(* Logix 5000 project; controller SX_V040001_C001 vendor 1 type 14 code 77 rev 16.22; software revision 16.04; part 18 of 35 *)
(* tags used below, declared in another part *)
   ALL_KINDS : INT[90];
   Basic : INT;
   DRIVE : INT[32];
   Drive_diff_rpm_real : REAL;
   Drive_set_prop_rpm_real : REAL;
   G_AOutput : DINT[8];
   G_DInput : DINT[3];
   G_DOutput : DINT[3];
   PARAMETER : INT[501];
   T_DELAY_COOLING_FAN : TIMER;
   T_DRIVE_START_WARN : TIMER;
   TEMP : INT[14];
(* MainProgram, continued *)

ROUTINE MainDriveFrequenc   (* ladder *)
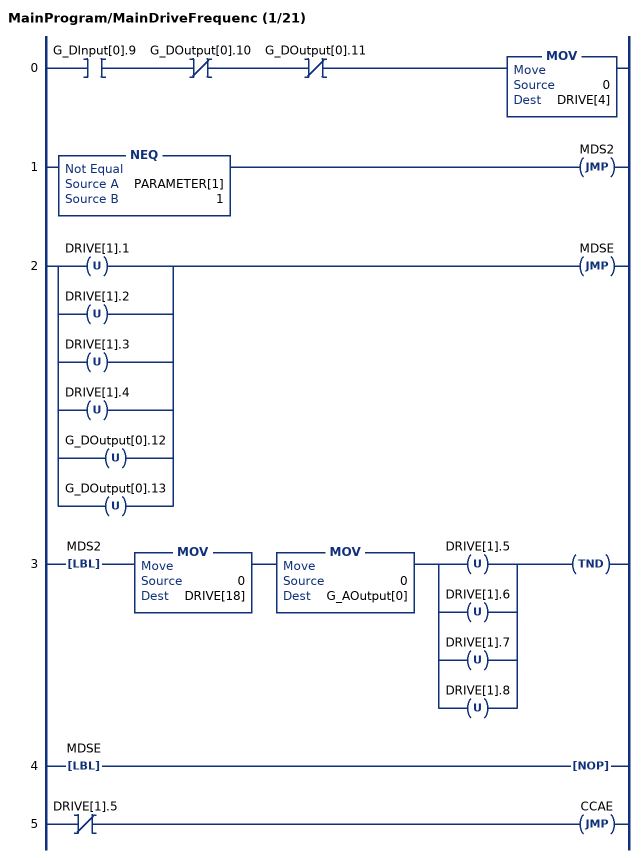
   0: XIC(G_DInput[0].9)XIO(G_DOutput[0].10)XIO(G_DOutput[0].11)MOV(0,DRIVE[4]);
   1: NEQ(PARAMETER[1],1)JMP(MDS2);
   2: [OTU(DRIVE[1].1) ,OTU(DRIVE[1].2) ,OTU(DRIVE[1].3) ,OTU(DRIVE[1].4) ,OTU(G_DOutput[0].12) ,OTU(G_DOutput[0].13) ]JMP(MDSE);
   3: LBL(MDS2)MOV(0,DRIVE[18])MOV(0,G_AOutput[0])[OTU(DRIVE[1].5) ,OTU(DRIVE[1].6) ,OTU(DRIVE[1].7) ,OTU(DRIVE[1].8) ]TND();
   4: LBL(MDSE)NOP();
   5: XIO(DRIVE[1].5)JMP(CCAE);
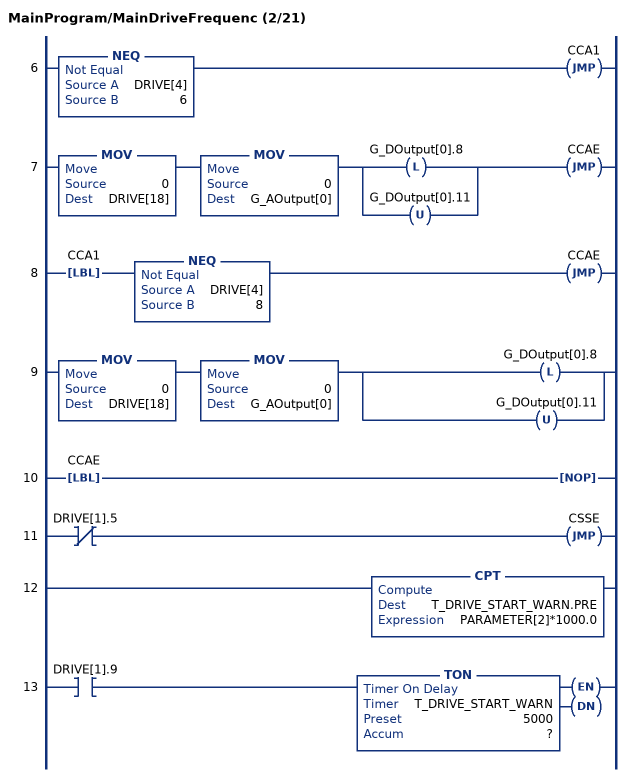
   6: NEQ(DRIVE[4],6)JMP(CCA1);
   7: MOV(0,DRIVE[18])MOV(0,G_AOutput[0])[OTL(G_DOutput[0].8) ,OTU(G_DOutput[0].11) ]JMP(CCAE);
   8: LBL(CCA1)NEQ(DRIVE[4],8)JMP(CCAE);
   9: MOV(0,DRIVE[18])MOV(0,G_AOutput[0])[OTL(G_DOutput[0].8) ,OTU(G_DOutput[0].11) ];
   10: LBL(CCAE)NOP();
   11: XIO(DRIVE[1].5)JMP(CSSE);
   12: CPT(T_DRIVE_START_WARN.PRE,PARAMETER[2]*1000.0);
   13: XIC(DRIVE[1].9)TON(T_DRIVE_START_WARN,?,?);
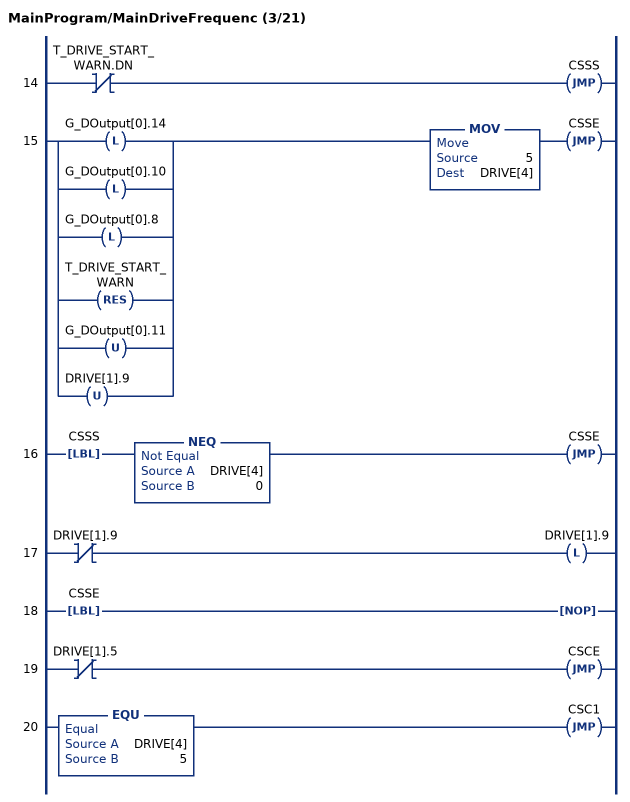
   14: XIO(T_DRIVE_START_WARN.DN)JMP(CSSS);
   15: [OTL(G_DOutput[0].14) ,OTL(G_DOutput[0].10) ,OTL(G_DOutput[0].8) ,RES(T_DRIVE_START_WARN) ,OTU(G_DOutput[0].11) ,OTU(DRIVE[1].9) ]MOV(5,DRIVE[4])JMP(CSSE);
   16: LBL(CSSS)NEQ(DRIVE[4],0)JMP(CSSE);
   17: XIO(DRIVE[1].9)OTL(DRIVE[1].9);
   18: LBL(CSSE)NOP();
   19: XIO(DRIVE[1].5)JMP(CSCE);
   20: EQU(DRIVE[4],5)JMP(CSC1);
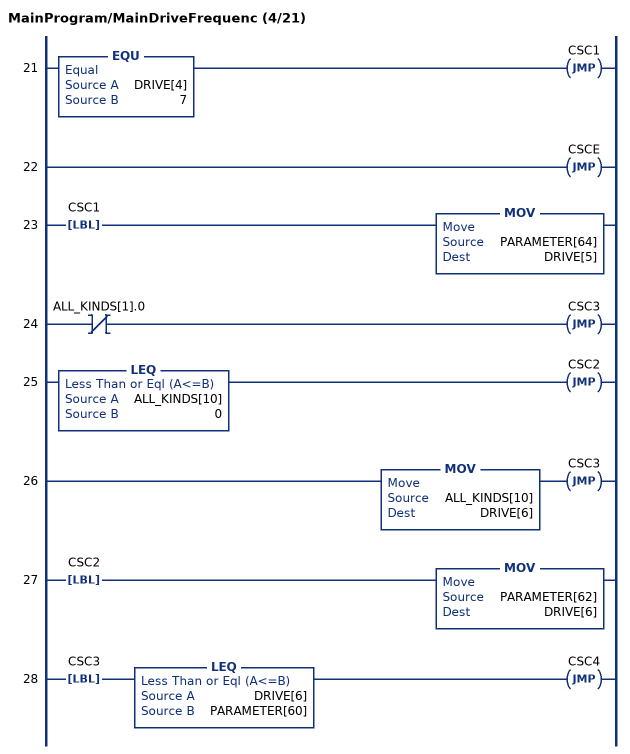
   21: EQU(DRIVE[4],7)JMP(CSC1);
   22: JMP(CSCE);
   23: LBL(CSC1)MOV(PARAMETER[64],DRIVE[5]);
   24: XIO(ALL_KINDS[1].0)JMP(CSC3);
   25: LEQ(ALL_KINDS[10],0)JMP(CSC2);
   26: MOV(ALL_KINDS[10],DRIVE[6])JMP(CSC3);
   27: LBL(CSC2)MOV(PARAMETER[62],DRIVE[6]);
   28: LBL(CSC3)LEQ(DRIVE[6],PARAMETER[60])JMP(CSC4);
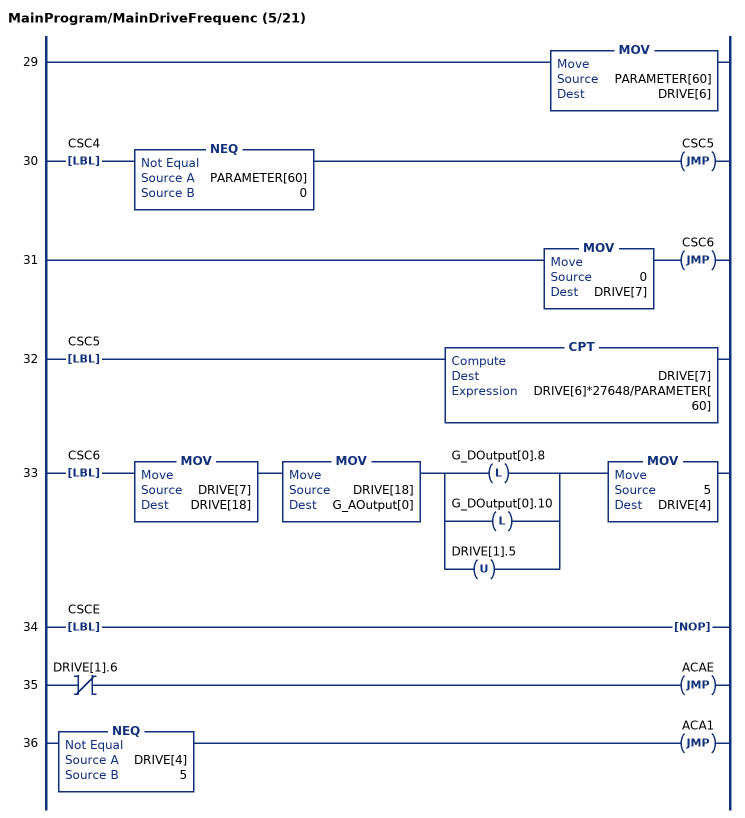
   29: MOV(PARAMETER[60],DRIVE[6]);
   30: LBL(CSC4)NEQ(PARAMETER[60],0)JMP(CSC5);
   31: MOV(0,DRIVE[7])JMP(CSC6);
   32: LBL(CSC5)CPT(DRIVE[7],DRIVE[6]*27648/PARAMETER[60]);
   33: LBL(CSC6)MOV(DRIVE[7],DRIVE[18])MOV(DRIVE[18],G_AOutput[0])[OTL(G_DOutput[0].8) ,OTL(G_DOutput[0].10) ,OTU(DRIVE[1].5) ]MOV(5,DRIVE[4]);
   34: LBL(CSCE)NOP();
   35: XIO(DRIVE[1].6)JMP(ACAE);
   36: NEQ(DRIVE[4],5)JMP(ACA1);
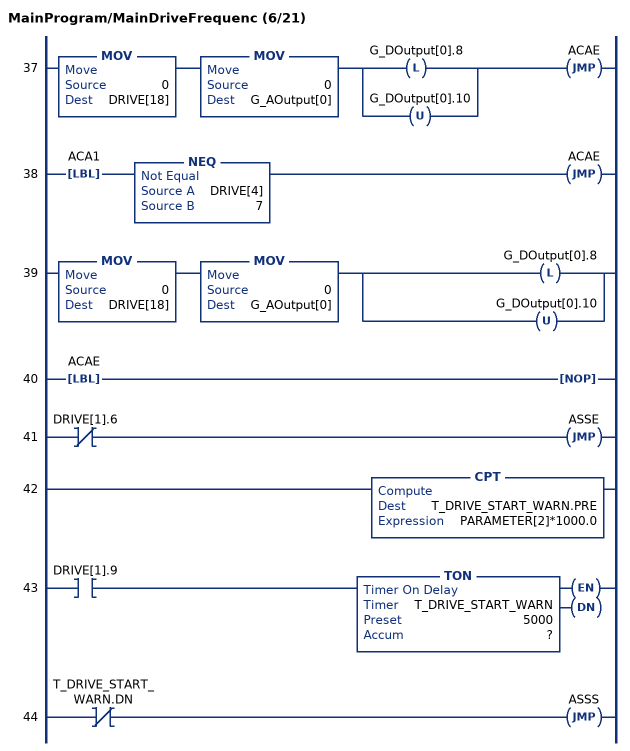
   37: MOV(0,DRIVE[18])MOV(0,G_AOutput[0])[OTL(G_DOutput[0].8) ,OTU(G_DOutput[0].10) ]JMP(ACAE);
   38: LBL(ACA1)NEQ(DRIVE[4],7)JMP(ACAE);
   39: MOV(0,DRIVE[18])MOV(0,G_AOutput[0])[OTL(G_DOutput[0].8) ,OTU(G_DOutput[0].10) ];
   40: LBL(ACAE)NOP();
   41: XIO(DRIVE[1].6)JMP(ASSE);
   42: CPT(T_DRIVE_START_WARN.PRE,PARAMETER[2]*1000.0);
   43: XIC(DRIVE[1].9)TON(T_DRIVE_START_WARN,?,?);
   44: XIO(T_DRIVE_START_WARN.DN)JMP(ASSS);
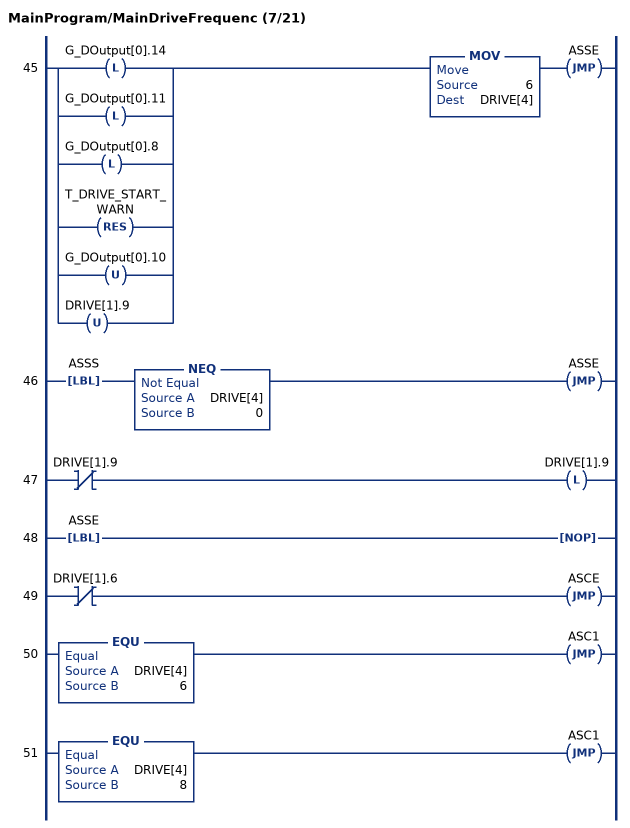
   45: [OTL(G_DOutput[0].14) ,OTL(G_DOutput[0].11) ,OTL(G_DOutput[0].8) ,RES(T_DRIVE_START_WARN) ,OTU(G_DOutput[0].10) ,OTU(DRIVE[1].9) ]MOV(6,DRIVE[4])JMP(ASSE);
   46: LBL(ASSS)NEQ(DRIVE[4],0)JMP(ASSE);
   47: XIO(DRIVE[1].9)OTL(DRIVE[1].9);
   48: LBL(ASSE)NOP();
   49: XIO(DRIVE[1].6)JMP(ASCE);
   50: EQU(DRIVE[4],6)JMP(ASC1);
   51: EQU(DRIVE[4],8)JMP(ASC1);
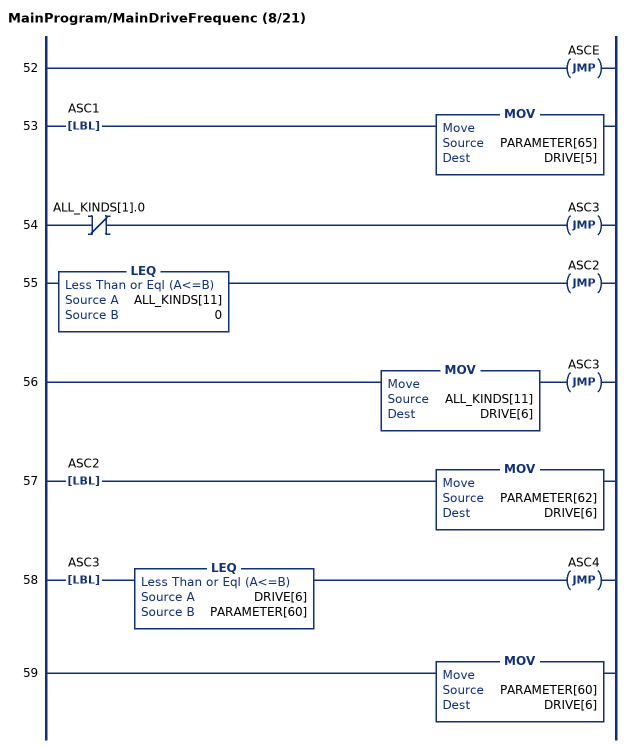
   52: JMP(ASCE);
   53: LBL(ASC1)MOV(PARAMETER[65],DRIVE[5]);
   54: XIO(ALL_KINDS[1].0)JMP(ASC3);
   55: LEQ(ALL_KINDS[11],0)JMP(ASC2);
   56: MOV(ALL_KINDS[11],DRIVE[6])JMP(ASC3);
   57: LBL(ASC2)MOV(PARAMETER[62],DRIVE[6]);
   58: LBL(ASC3)LEQ(DRIVE[6],PARAMETER[60])JMP(ASC4);
   59: MOV(PARAMETER[60],DRIVE[6]);
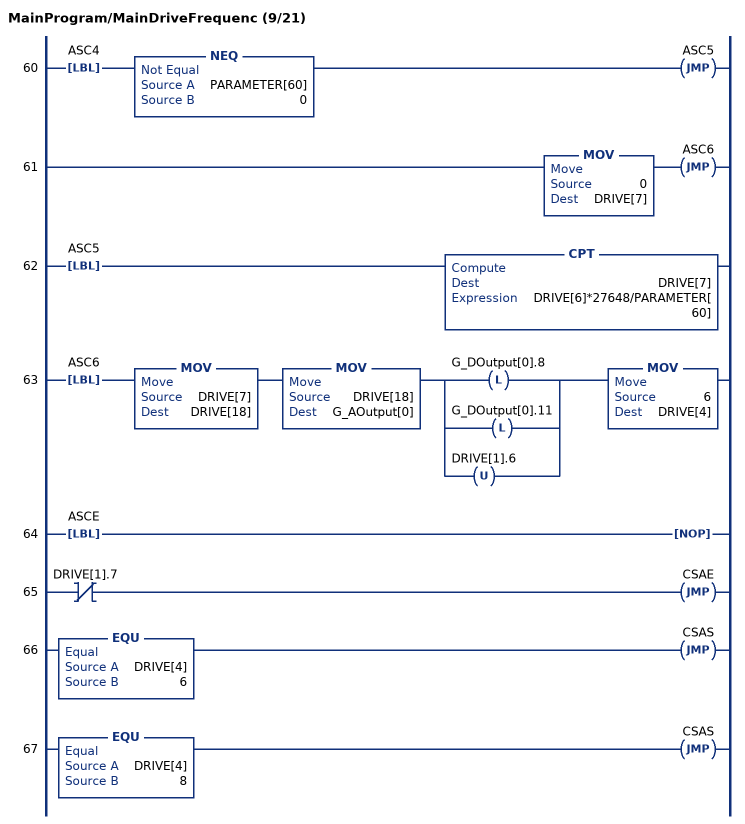
   60: LBL(ASC4)NEQ(PARAMETER[60],0)JMP(ASC5);
   61: MOV(0,DRIVE[7])JMP(ASC6);
   62: LBL(ASC5)CPT(DRIVE[7],DRIVE[6]*27648/PARAMETER[60]);
   63: LBL(ASC6)MOV(DRIVE[7],DRIVE[18])MOV(DRIVE[18],G_AOutput[0])[OTL(G_DOutput[0].8) ,OTL(G_DOutput[0].11) ,OTU(DRIVE[1].6) ]MOV(6,DRIVE[4]);
   64: LBL(ASCE)NOP();
   65: XIO(DRIVE[1].7)JMP(CSAE);
   66: EQU(DRIVE[4],6)JMP(CSAS);
   67: EQU(DRIVE[4],8)JMP(CSAS);
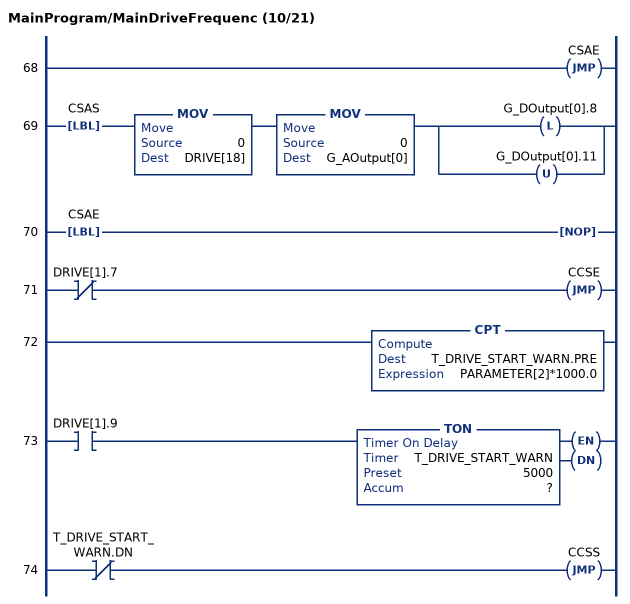
   68: JMP(CSAE);
   69: LBL(CSAS)MOV(0,DRIVE[18])MOV(0,G_AOutput[0])[OTL(G_DOutput[0].8) ,OTU(G_DOutput[0].11) ];
   70: LBL(CSAE)NOP();
   71: XIO(DRIVE[1].7)JMP(CCSE);
   72: CPT(T_DRIVE_START_WARN.PRE,PARAMETER[2]*1000.0);
   73: XIC(DRIVE[1].9)TON(T_DRIVE_START_WARN,?,?);
   74: XIO(T_DRIVE_START_WARN.DN)JMP(CCSS);
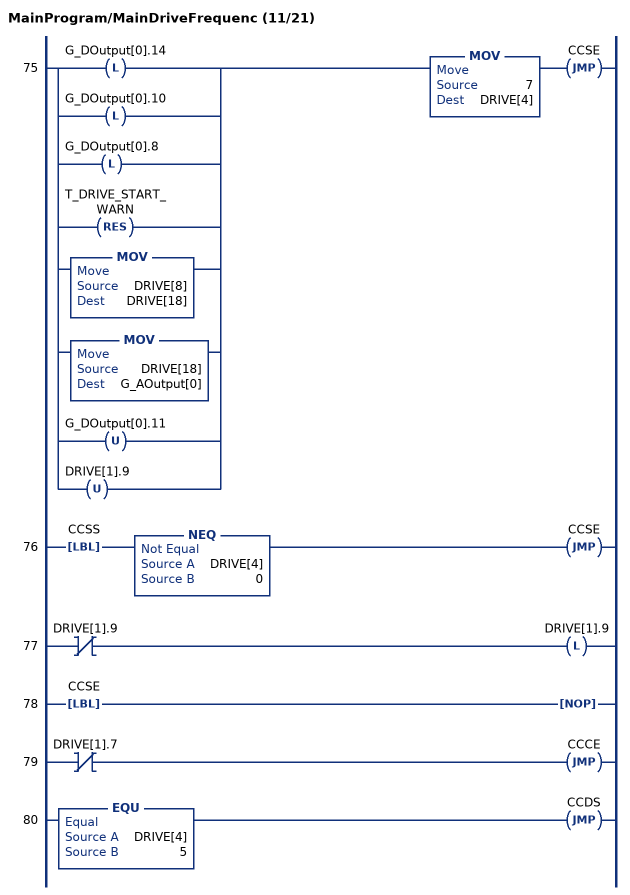
   75: [OTL(G_DOutput[0].14) ,OTL(G_DOutput[0].10) ,OTL(G_DOutput[0].8) ,RES(T_DRIVE_START_WARN) ,MOV(DRIVE[8],DRIVE[18]) ,MOV(DRIVE[18],G_AOutput[0]) ,OTU(G_DOutput[0].11) ,OTU(DRIVE[1].9) ]MOV(7,DRIVE[4])JMP(CCSE);
   76: LBL(CCSS)NEQ(DRIVE[4],0)JMP(CCSE);
   77: XIO(DRIVE[1].9)OTL(DRIVE[1].9);
   78: LBL(CCSE)NOP();
   79: XIO(DRIVE[1].7)JMP(CCCE);
   80: EQU(DRIVE[4],5)JMP(CCDS);
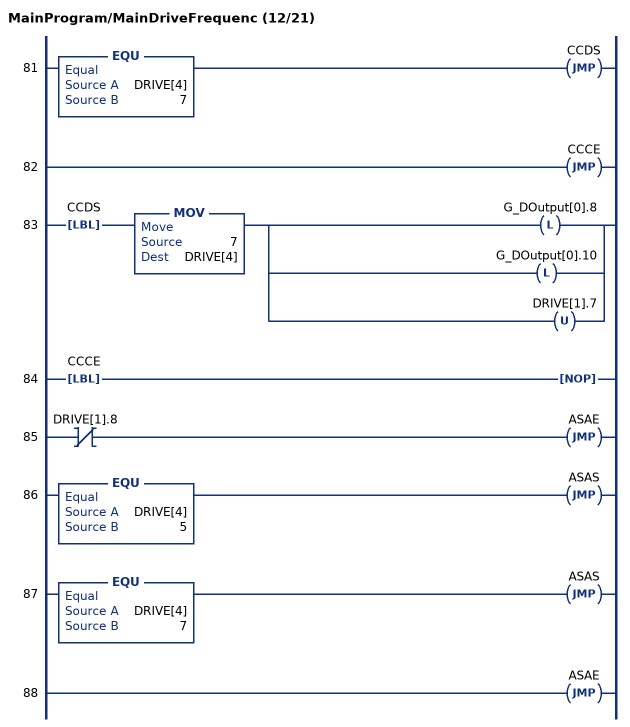
   81: EQU(DRIVE[4],7)JMP(CCDS);
   82: JMP(CCCE);
   83: LBL(CCDS)MOV(7,DRIVE[4])[OTL(G_DOutput[0].8) ,OTL(G_DOutput[0].10) ,OTU(DRIVE[1].7) ];
   84: LBL(CCCE)NOP();
   85: XIO(DRIVE[1].8)JMP(ASAE);
   86: EQU(DRIVE[4],5)JMP(ASAS);
   87: EQU(DRIVE[4],7)JMP(ASAS);
   88: JMP(ASAE);
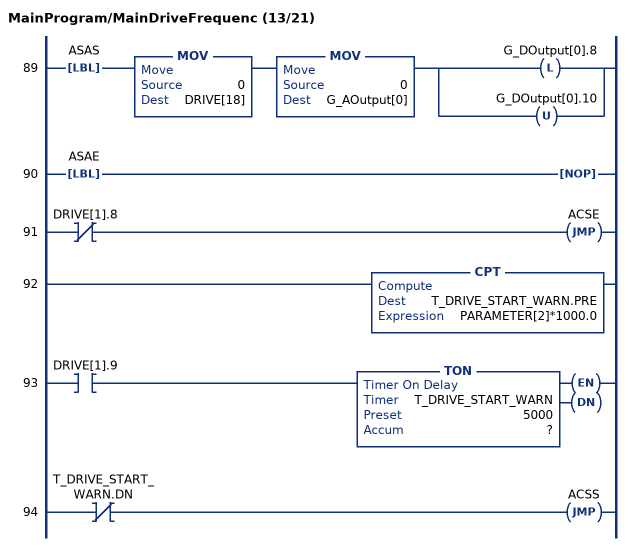
   89: LBL(ASAS)MOV(0,DRIVE[18])MOV(0,G_AOutput[0])[OTL(G_DOutput[0].8) ,OTU(G_DOutput[0].10) ];
   90: LBL(ASAE)NOP();
   91: XIO(DRIVE[1].8)JMP(ACSE);
   92: CPT(T_DRIVE_START_WARN.PRE,PARAMETER[2]*1000.0);
   93: XIC(DRIVE[1].9)TON(T_DRIVE_START_WARN,?,?);
   94: XIO(T_DRIVE_START_WARN.DN)JMP(ACSS);
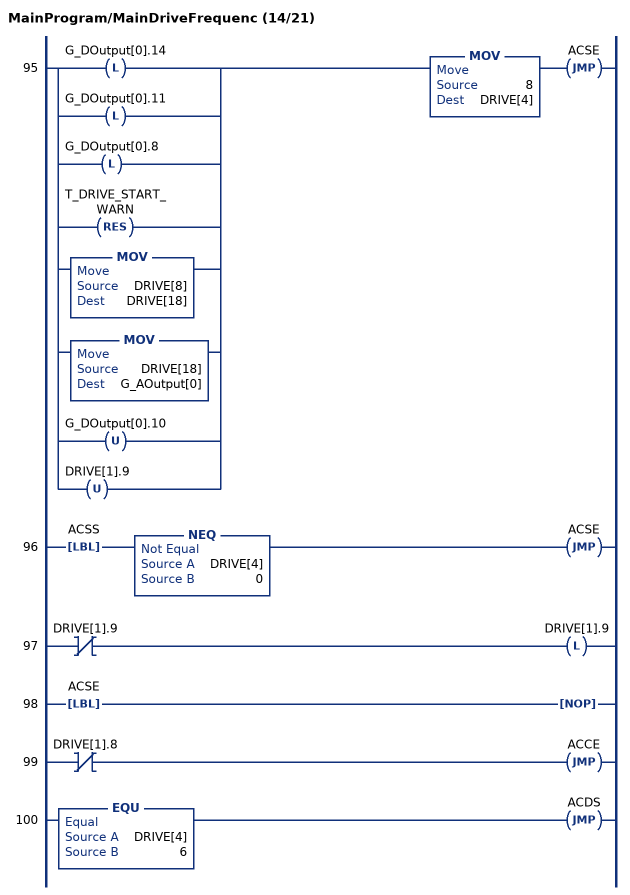
   95: [OTL(G_DOutput[0].14) ,OTL(G_DOutput[0].11) ,OTL(G_DOutput[0].8) ,RES(T_DRIVE_START_WARN) ,MOV(DRIVE[8],DRIVE[18]) ,MOV(DRIVE[18],G_AOutput[0]) ,OTU(G_DOutput[0].10) ,OTU(DRIVE[1].9) ]MOV(8,DRIVE[4])JMP(ACSE);
   96: LBL(ACSS)NEQ(DRIVE[4],0)JMP(ACSE);
   97: XIO(DRIVE[1].9)OTL(DRIVE[1].9);
   98: LBL(ACSE)NOP();
   99: XIO(DRIVE[1].8)JMP(ACCE);
   100: EQU(DRIVE[4],6)JMP(ACDS);
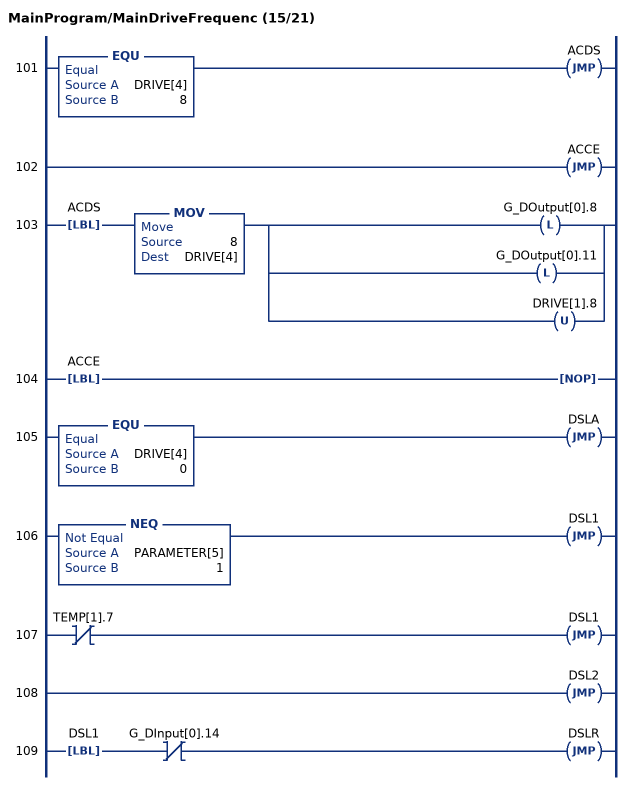
   101: EQU(DRIVE[4],8)JMP(ACDS);
   102: JMP(ACCE);
   103: LBL(ACDS)MOV(8,DRIVE[4])[OTL(G_DOutput[0].8) ,OTL(G_DOutput[0].11) ,OTU(DRIVE[1].8) ];
   104: LBL(ACCE)NOP();
   105: EQU(DRIVE[4],0)JMP(DSLA);
   106: NEQ(PARAMETER[5],1)JMP(DSL1);
   107: XIO(TEMP[1].7)JMP(DSL1);
   108: JMP(DSL2);
   109: LBL(DSL1)XIO(G_DInput[0].14)JMP(DSLR);
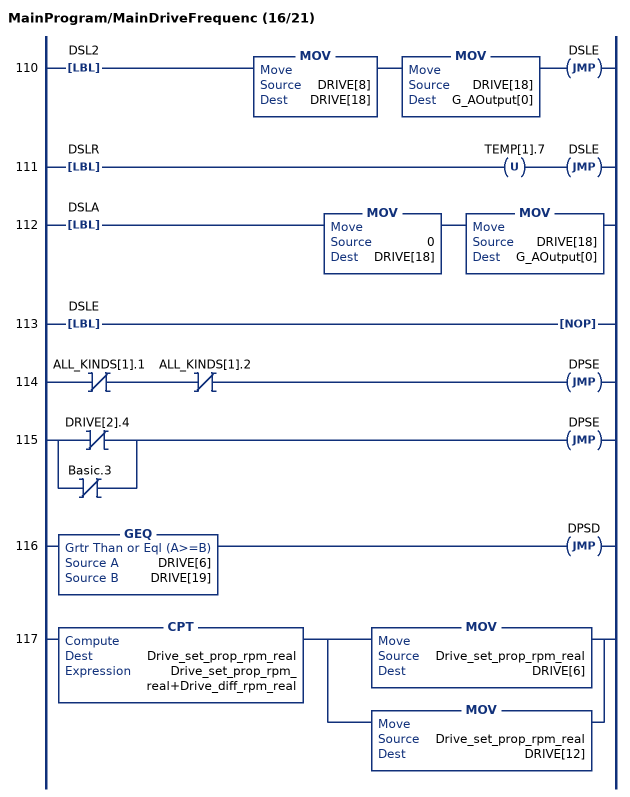
   110: LBL(DSL2)MOV(DRIVE[8],DRIVE[18])MOV(DRIVE[18],G_AOutput[0])JMP(DSLE);
   111: LBL(DSLR)OTU(TEMP[1].7)JMP(DSLE);
   112: LBL(DSLA)MOV(0,DRIVE[18])MOV(DRIVE[18],G_AOutput[0]);
   113: LBL(DSLE)NOP();
   114: XIO(ALL_KINDS[1].1)XIO(ALL_KINDS[1].2)JMP(DPSE);
   115: [XIO(DRIVE[2].4) ,XIO(Basic.3) ]JMP(DPSE);
   116: GEQ(DRIVE[6],DRIVE[19])JMP(DPSD);
   117: CPT(Drive_set_prop_rpm_real,Drive_set_prop_rpm_real+Drive_diff_rpm_real)[MOV(Drive_set_prop_rpm_real,DRIVE[6]) ,MOV(Drive_set_prop_rpm_real,DRIVE[12]) ];
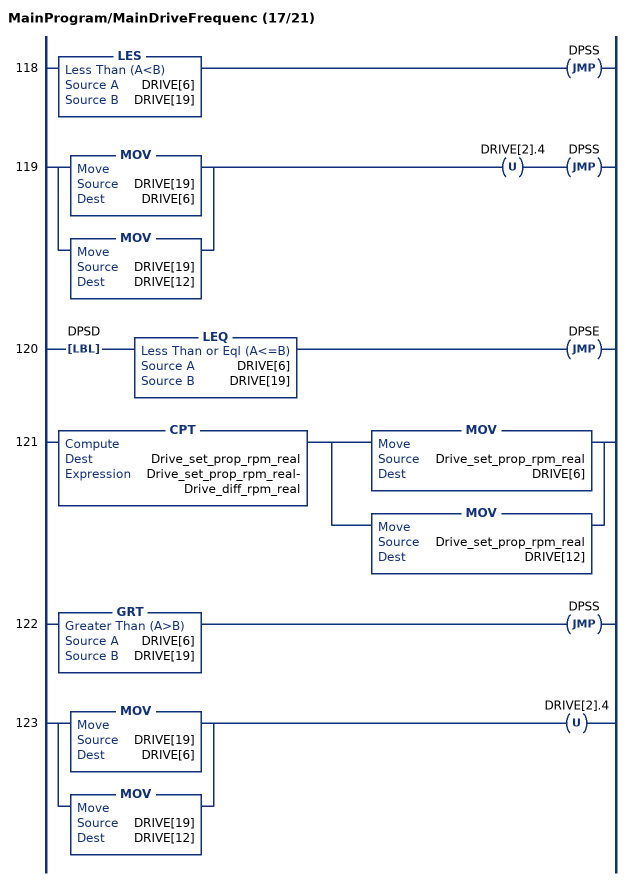
   118: LES(DRIVE[6],DRIVE[19])JMP(DPSS);
   119: [MOV(DRIVE[19],DRIVE[6]) ,MOV(DRIVE[19],DRIVE[12]) ]OTU(DRIVE[2].4)JMP(DPSS);
   120: LBL(DPSD)LEQ(DRIVE[6],DRIVE[19])JMP(DPSE);
   121: CPT(Drive_set_prop_rpm_real,Drive_set_prop_rpm_real-Drive_diff_rpm_real)[MOV(Drive_set_prop_rpm_real,DRIVE[6]) ,MOV(Drive_set_prop_rpm_real,DRIVE[12]) ];
   122: GRT(DRIVE[6],DRIVE[19])JMP(DPSS);
   123: [MOV(DRIVE[19],DRIVE[6]) ,MOV(DRIVE[19],DRIVE[12]) ]OTU(DRIVE[2].4);
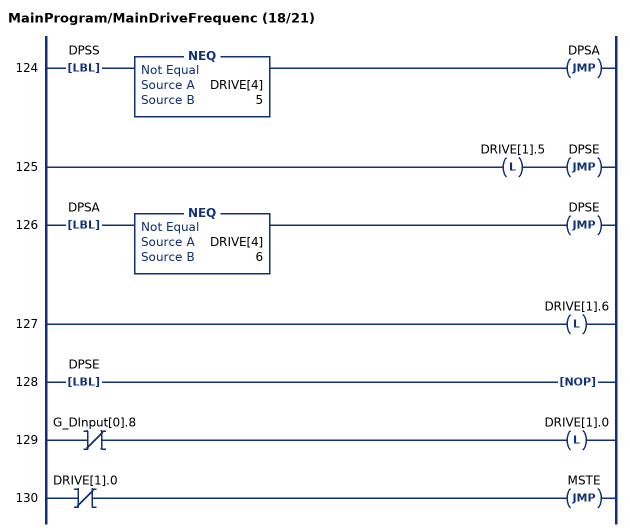
   124: LBL(DPSS)NEQ(DRIVE[4],5)JMP(DPSA);
   125: OTL(DRIVE[1].5)JMP(DPSE);
   126: LBL(DPSA)NEQ(DRIVE[4],6)JMP(DPSE);
   127: OTL(DRIVE[1].6);
   128: LBL(DPSE)NOP();
   129: XIO(G_DInput[0].8)OTL(DRIVE[1].0);
   130: XIO(DRIVE[1].0)JMP(MSTE);
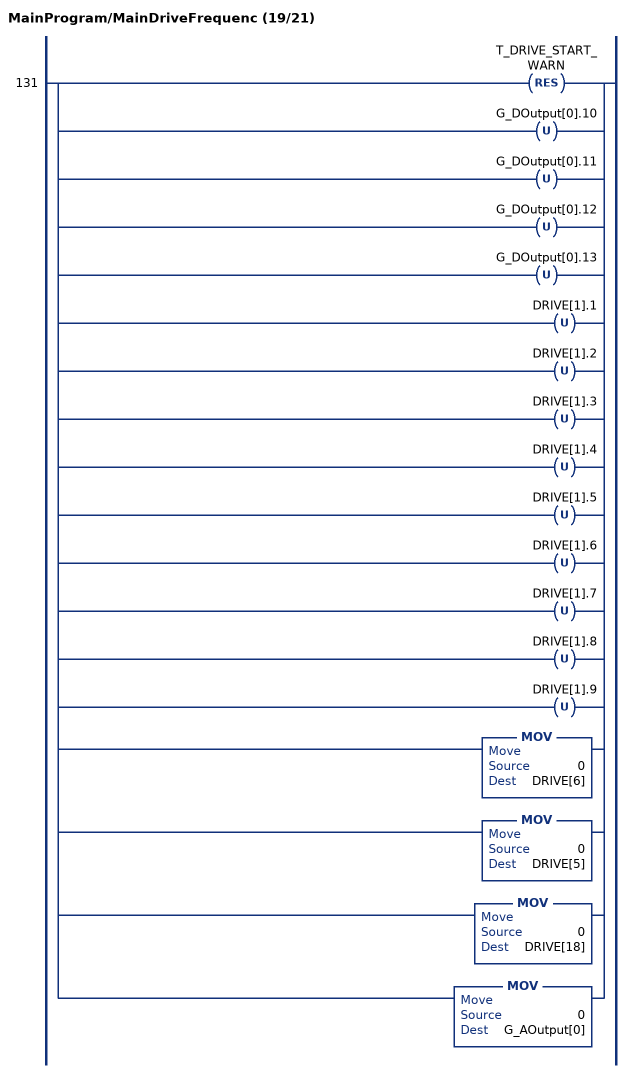
   131: [RES(T_DRIVE_START_WARN) ,OTU(G_DOutput[0].10) ,OTU(G_DOutput[0].11) ,OTU(G_DOutput[0].12) ,OTU(G_DOutput[0].13) ,OTU(DRIVE[1].1) ,OTU(DRIVE[1].2) ,OTU(DRIVE[1].3) ,OTU(DRIVE[1].4) ,OTU(DRIVE[1].5) ,OTU(DRIVE[1].6) ,OTU(DRIVE[1].7) ,OTU(DRIVE[1].8) ,OTU(DRIVE[1].9) ,MOV(0,DRIVE[6]) ,MOV(0,DRIVE[5]) ,MOV(0,DRIVE[18]) ,MOV(0,G_AOutput[0]) ];
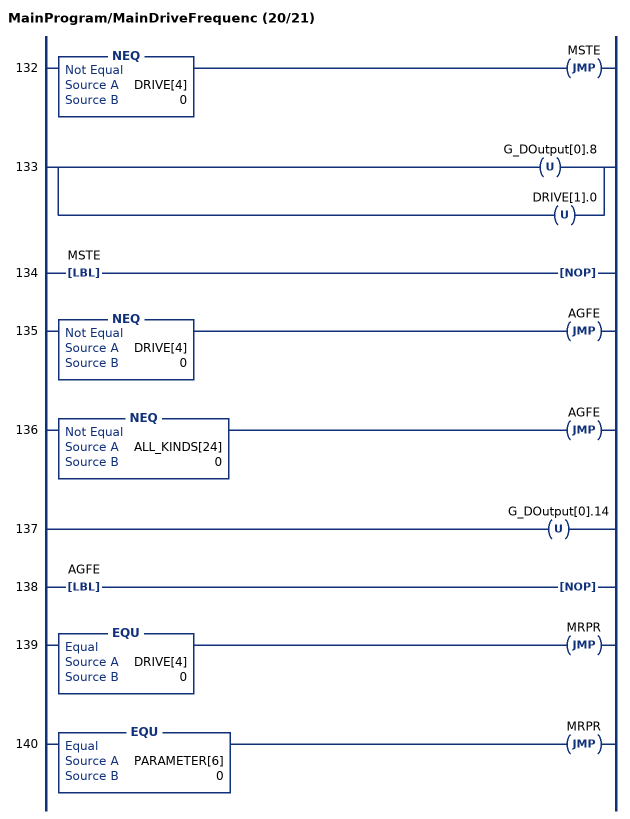
   132: NEQ(DRIVE[4],0)JMP(MSTE);
   133: [OTU(G_DOutput[0].8) ,OTU(DRIVE[1].0) ];
   134: LBL(MSTE)NOP();
   135: NEQ(DRIVE[4],0)JMP(AGFE);
   136: NEQ(ALL_KINDS[24],0)JMP(AGFE);
   137: OTU(G_DOutput[0].14);
   138: LBL(AGFE)NOP();
   139: EQU(DRIVE[4],0)JMP(MRPR);
   140: EQU(PARAMETER[6],0)JMP(MRPR);
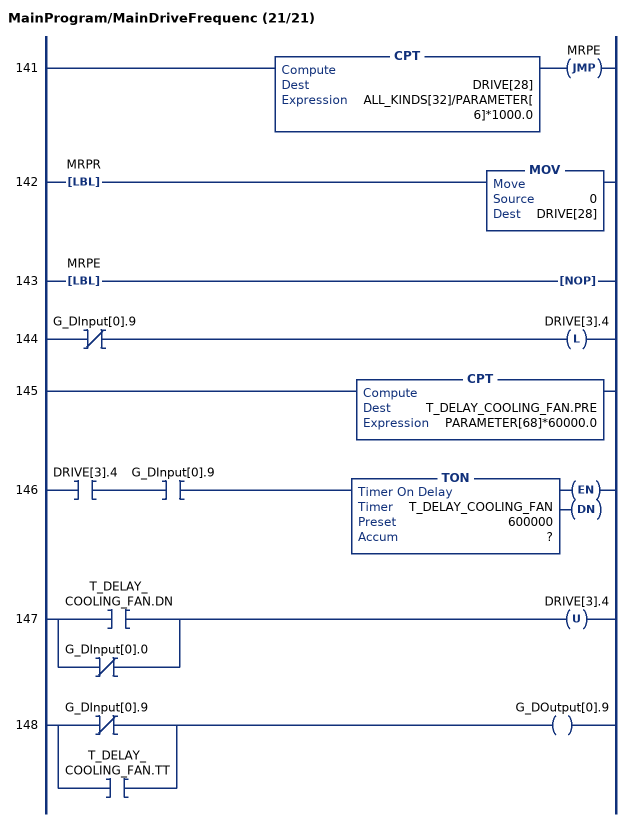
   141: CPT(DRIVE[28],ALL_KINDS[32]/PARAMETER[6]*1000.0)JMP(MRPE);
   142: LBL(MRPR)MOV(0,DRIVE[28]);
   143: LBL(MRPE)NOP();
   144: XIO(G_DInput[0].9)OTL(DRIVE[3].4);
   145: CPT(T_DELAY_COOLING_FAN.PRE,PARAMETER[68]*60000.0);
   146: XIC(DRIVE[3].4)XIC(G_DInput[0].9)TON(T_DELAY_COOLING_FAN,?,?);
   147: [XIC(T_DELAY_COOLING_FAN.DN) ,XIO(G_DInput[0].0) ]OTU(DRIVE[3].4);
   148: [XIO(G_DInput[0].9) ,XIC(T_DELAY_COOLING_FAN.TT) ]OTE(G_DOutput[0].9);
END_ROUTINE
